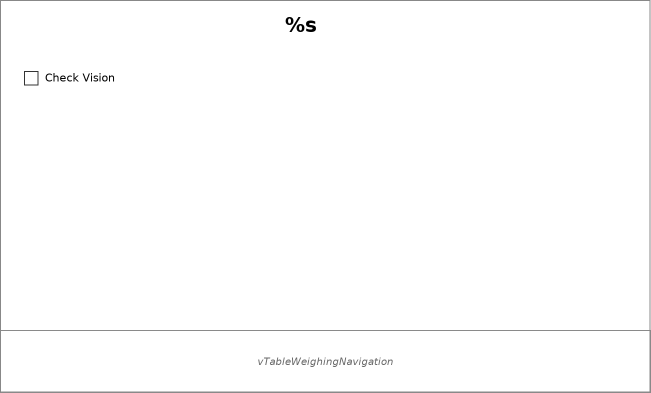
VISUALIZATION vTableWeighingVision  // 651x393
VAR_IN_OUT
	fbStation:FB_WeighingStation;
	fbTableControl: FB_TableControl;
END_VAR
    Rectangle (0,0 650x392)
    Rectangle (226,10 150x30), "%s", text variable: fbStation.sStationName
    Frame (0,330 651x63)
        shows vTableWeighingNavigation(fbTableControl := fbTableControl)
    Checkbox (22,63 150x30), "Check Vision", variable: fbStation.stSettings.bCameraCheck
END_VISUALIZATION

(* stored: Version 1.1.0.1, ProductVersion 3.1.4024.15
   Visu vTableWeighingVision: Id {da3b69c6-1059-4496-8601-c1829e9a3568} *)
